///  Skill variables inside DUT_TASK
TYPE DUT_SKILL :
STRUCT
	///Name assigned for the process tool
	AssignedModuleName: STRING[80];
	///ID assigned for the process tool
	AssignedModuleID: UINT;
	///Position assigned for the process tool
	AssignedModulePosition: LREAL;
	///Free to use = TRUE, busy to use =FALSE
	Dummy: BOOL := TRUE;
	///Identification number of the skill
	ID: UINT;
	///Name of the skill
	Name: STRING[80];
	// State of the skill
	State: INT;
	///Range of parameters
	Parameter: ARRAY[0..ParameterCnt] OF DUT_PARAMETER;
END_STRUCT
END_TYPE

(* stored: Version 1.1.0.1, ProductVersion 3.1.0.25
   DUT DUT_SKILL: Id {3c1f9679-e16c-44a3-8cf2-e8fb30cc40c5} *)
